# EPICS substitutions: odmApp/Db/odm-test.substitutions
file pilz-plc-bi-table9seg1.template
{
	pattern
	{dtype, areapos,  attribute,     description,                       port,    bit,   zname,         oname,                 zsv,        osv, plc           }

#################################################################### ODM PILZ PLC ##########################################################################

	{ ODM, CR1:1:0,  FAULT,         "C1 West Oxigraf Ch0 Real",       ODM_RD,      7,   OK,            FAULT,               NO_ALARM,   MAJOR, PLC:CP00:OD01 }
	{ ODM, CR1:1:0,  FAULT_LTH,     "C1 West Oxigraf Ch0 Latch",      ODM_RD,      6,   OK,            FAULT,               NO_ALARM,   MAJOR, PLC:CP00:OD01 }
	{ ODM, CR1:1:1,  FAULT,         "C1 West Oxigraf Ch1 Real",       ODM_RD,      5,   OK,            FAULT,               NO_ALARM,   MAJOR, PLC:CP00:OD01 }
	{ ODM, CR1:1:1,  FAULT_LTH,     "C1 West Oxigraf Ch1 Latch",      ODM_RD,      4,   OK,            FAULT,               NO_ALARM,   MAJOR, PLC:CP00:OD01 }
	{ ODM, CR1:1:2,  FAULT,         "C1 West Oxigraf Ch2 Real",       ODM_RD,      3,   OK,            FAULT,               NO_ALARM,   MAJOR, PLC:CP00:OD01 }
	{ ODM, CR1:1:2,  FAULT_LTH,     "C1 West Oxigraf Ch2 Latch",      ODM_RD,      2,   OK,            FAULT,               NO_ALARM,   MAJOR, PLC:CP00:OD01 }
	{ ODM, CR1:1:3,  FAULT,         "C1 West Oxigraf Ch3 Real",       ODM_RD,      1,   OK,            FAULT,               NO_ALARM,   MAJOR, PLC:CP00:OD01 }
	{ ODM, CR1:1:3,  FAULT_LTH,     "C1 West Oxigraf Ch3 Latch",      ODM_RD,      0,   OK,            FAULT,               NO_ALARM,   MAJOR, PLC:CP00:OD01 }
	{ ODM, CR1:2:0,  FAULT,         "C1 East Oxigraf Ch0 Real",       ODM_RD,      15,  OK,            FAULT,               NO_ALARM,   MAJOR, PLC:CP00:OD01 }
	{ ODM, CR1:2:0,  FAULT_LTH,     "C1 East Oxigraf Ch0 Latch",      ODM_RD,      14,  OK,            FAULT,               NO_ALARM,   MAJOR, PLC:CP00:OD01 }
	{ ODM, CR1:2:1,  FAULT,         "C1 East Oxigraf Ch1 Real",       ODM_RD,      13,  OK,            FAULT,               NO_ALARM,   MAJOR, PLC:CP00:OD01 }
	{ ODM, CR1:2:1,  FAULT_LTH,     "C1 East Oxigraf Ch1 Latch",      ODM_RD,      12,  OK,            FAULT,               NO_ALARM,   MAJOR, PLC:CP00:OD01 }
	{ ODM, CR1:2:2,  FAULT,         "C1 East Oxigraf Ch2 Real",       ODM_RD,      11,  OK,            FAULT,               NO_ALARM,   MAJOR, PLC:CP00:OD01 }
	{ ODM, CR1:2:2,  FAULT_LTH,     "C1 East Oxigraf Ch2 Latch",      ODM_RD,      10,  OK,            FAULT,               NO_ALARM,   MAJOR, PLC:CP00:OD01 }
	{ ODM, CR1:2:3,  FAULT,         "C1 East Oxigraf Ch3 Real",       ODM_RD,      9,   OK,            FAULT,               NO_ALARM,   MAJOR, PLC:CP00:OD01 }
	{ ODM, CR1:2:3,  FAULT_LTH,     "C1 East Oxigraf Ch3 Latch",      ODM_RD,      8,   OK,            FAULT,               NO_ALARM,   MAJOR, PLC:CP00:OD01 }
	{ ODM, CR1:1,    SYS_OK,        "C1 West Sys OK Real",            ODM_RD,      23,  OK,            FAULT,               NO_ALARM,   MAJOR, PLC:CP00:OD01 }
	{ ODM, CR1:1,    SYS_OK_LTH,    "C1 West Sys OK Latch",           ODM_RD,      22,  OK,            FAULT,               NO_ALARM,   MAJOR, PLC:CP00:OD01 }
	{ ODM, CR1:2,    SYS_OK,        "C1 East Sys OK Real",            ODM_RD,      21,  OK,            FAULT,               NO_ALARM,   MAJOR, PLC:CP00:OD01 }
	{ ODM, CR1:2,    SYS_OK_LTH,    "C1 East Sys OK Latch",           ODM_RD,      20,  OK,            FAULT,               NO_ALARM,   MAJOR, PLC:CP00:OD01 }
	{ ODM, CR0:1:0,  FAULT,         "CBR West Oxigraf Ch0 Real",      ODM_RD,      19,  OK,            FAULT,               NO_ALARM,   MAJOR, PLC:CP00:OD01 }
	{ ODM, CR0:1:0,  FAULT_LTH,     "CBR West Oxigraf Ch0 Latch",     ODM_RD,      18,  OK,            FAULT,               NO_ALARM,   MAJOR, PLC:CP00:OD01 }
	{ ODM, CR0:1:1,  FAULT,         "CBR West Oxigraf Ch1 Real",      ODM_RD,      17,  OK,            FAULT,               NO_ALARM,   MAJOR, PLC:CP00:OD01 }
	{ ODM, CR0:1:1,  FAULT_LTH,     "CBR West Oxigraf Ch1 Latch",     ODM_RD,      16,  OK,            FAULT,               NO_ALARM,   MAJOR, PLC:CP00:OD01 }
	{ ODM, CR0:1:2,  FAULT,         "CBR West Oxigraf Ch2 Real",      ODM_RD,      95,  OK,            FAULT,               NO_ALARM,   MAJOR, PLC:CP00:OD01 }
	{ ODM, CR0:1:2,  FAULT_LTH,     "CBR West Oxigraf Ch2 Latch",     ODM_RD,      94,  OK,            FAULT,               NO_ALARM,   MAJOR, PLC:CP00:OD01 }
	{ ODM, CR0:1:3,  FAULT,         "CBR West Oxigraf Ch3 Real",      ODM_RD,      93,  OK,            FAULT,               NO_ALARM,   MAJOR, PLC:CP00:OD01 }
	{ ODM, CR0:1:3,  FAULT_LTH,     "CBR West Oxigraf Ch3 Latch",     ODM_RD,      92,  OK,            FAULT,               NO_ALARM,   MAJOR, PLC:CP00:OD01 }
	{ ODM, CR0:2:0,  FAULT,         "CBR East Oxigraf Ch0 Real",      ODM_RD,      91,  OK,            FAULT,               NO_ALARM,   MAJOR, PLC:CP00:OD01 }
	{ ODM, CR0:2:0,  FAULT_LTH,     "CBR East Oxigraf Ch0 Latch",     ODM_RD,      90,  OK,            FAULT,               NO_ALARM,   MAJOR, PLC:CP00:OD01 }
	{ ODM, CR0:2:1,  FAULT,         "CBR East Oxigraf Ch1 Real",      ODM_RD,      89,  OK,            FAULT,               NO_ALARM,   MAJOR, PLC:CP00:OD01 }
	{ ODM, CR0:2:1,  FAULT_LTH,     "CBR East Oxigraf Ch1 Latch",     ODM_RD,      88,  OK,            FAULT,               NO_ALARM,   MAJOR, PLC:CP00:OD01 }
	{ ODM, CR0:2:2,  FAULT,         "CBR East Oxigraf Ch2 Real",      ODM_RD,      103, OK,            FAULT,               NO_ALARM,   MAJOR, PLC:CP00:OD01 }
	{ ODM, CR0:2:2,  FAULT_LTH,     "CBR East Oxigraf Ch2 Latch",     ODM_RD,      102, OK,            FAULT,               NO_ALARM,   MAJOR, PLC:CP00:OD01 }
	{ ODM, CR0:2:3,  FAULT,         "CBR East Oxigraf Ch3 Real",      ODM_RD,      101, OK,            FAULT,               NO_ALARM,   MAJOR, PLC:CP00:OD01 }
	{ ODM, CR0:2:3,  FAULT_LTH,     "CBR East Oxigraf Ch3 Latch",     ODM_RD,      100, OK,            FAULT,               NO_ALARM,   MAJOR, PLC:CP00:OD01 }
	{ ODM, CR0:1,    SYS_OK,        "CBR West Sys OK Real",           ODM_RD,      99,  OK,            FAULT,               NO_ALARM,   MAJOR, PLC:CP00:OD01 }
	{ ODM, CR0:1,    SYS_OK_LTH,    "CBR West Sys OK Latch",          ODM_RD,      98,  OK,            FAULT,               NO_ALARM,   MAJOR, PLC:CP00:OD01 }
	{ ODM, CR0:2,    SYS_OK,        "CBR East Sys OK Real",           ODM_RD,      97,  OK,            FAULT,               NO_ALARM,   MAJOR, PLC:CP00:OD01 }
	{ ODM, CR0:2,    SYS_OK_LTH,    "CBR East Sys OK Latch",          ODM_RD,      96,  OK,            FAULT,               NO_ALARM,   MAJOR, PLC:CP00:OD01 }
	{ ODM, CR2:1:0,  FAULT,         "C2 West Oxigraf Ch0 Real",       ODM_RD,      111, OK,            FAULT,               NO_ALARM,   MAJOR, PLC:CP00:OD01 }
	{ ODM, CR2:1:0,  FAULT_LTH,     "C2 West Oxigraf Ch0 Latch",      ODM_RD,      110, OK,            FAULT,               NO_ALARM,   MAJOR, PLC:CP00:OD01 }
	{ ODM, CR2:1:1,  FAULT,         "C2 West Oxigraf Ch1 Real",       ODM_RD,      109, OK,            FAULT,               NO_ALARM,   MAJOR, PLC:CP00:OD01 }
	{ ODM, CR2:1:1,  FAULT_LTH,     "C2 West Oxigraf Ch1 Latch",      ODM_RD,      108, OK,            FAULT,               NO_ALARM,   MAJOR, PLC:CP00:OD01 }
	{ ODM, CR2:1:2,  FAULT,         "C2 West Oxigraf Ch2 Real",       ODM_RD,      107, OK,            FAULT,               NO_ALARM,   MAJOR, PLC:CP00:OD01 }
	{ ODM, CR2:1:2,  FAULT_LTH,     "C2 West Oxigraf Ch2 Latch",      ODM_RD,      106, OK,            FAULT,               NO_ALARM,   MAJOR, PLC:CP00:OD01 }
	{ ODM, CR2:1:3,  FAULT,         "C2 West Oxigraf Ch3 Real",       ODM_RD,      105, OK,            FAULT,               NO_ALARM,   MAJOR, PLC:CP00:OD01 }
	{ ODM, CR2:1:3,  FAULT_LTH,     "C2 West Oxigraf Ch3 Latch",      ODM_RD,      104, OK,            FAULT,               NO_ALARM,   MAJOR, PLC:CP00:OD01 }
	{ ODM, CR2:2:0,  FAULT,         "C2 East Oxigraf Ch0 Real",       ODM_RD,      119, OK,            FAULT,               NO_ALARM,   MAJOR, PLC:CP00:OD01 }
	{ ODM, CR2:2:0,  FAULT_LTH,     "C2 East Oxigraf Ch0 Latch",      ODM_RD,      118, OK,            FAULT,               NO_ALARM,   MAJOR, PLC:CP00:OD01 }
	{ ODM, CR2:2:1,  FAULT,         "C2 East Oxigraf Ch1 Real",       ODM_RD,      117, OK,            FAULT,               NO_ALARM,   MAJOR, PLC:CP00:OD01 }
	{ ODM, CR2:2:1,  FAULT_LTH,     "C2 East Oxigraf Ch1 Latch",      ODM_RD,      116, OK,            FAULT,               NO_ALARM,   MAJOR, PLC:CP00:OD01 }
	{ ODM, CR2:2:2,  FAULT,         "C2 East Oxigraf Ch2 Real",       ODM_RD,      115, OK,            FAULT,               NO_ALARM,   MAJOR, PLC:CP00:OD01 }
	{ ODM, CR2:2:2,  FAULT_LTH,     "C2 East Oxigraf Ch2 Latch",      ODM_RD,      114, OK,            FAULT,               NO_ALARM,   MAJOR, PLC:CP00:OD01 }
	{ ODM, CR2:2:3,  FAULT,         "C2 East Oxigraf Ch3 Real",       ODM_RD,      113, OK,            FAULT,               NO_ALARM,   MAJOR, PLC:CP00:OD01 }
	{ ODM, CR2:2:3,  FAULT_LTH,     "C2 East Oxigraf Ch3 Latch",      ODM_RD,      112, OK,            FAULT,               NO_ALARM,   MAJOR, PLC:CP00:OD01 }
	{ ODM, CR2:1,    SYS_OK,        "C2 West Sys OK Real",            ODM_RD,      127, OK,            FAULT,               NO_ALARM,   MAJOR, PLC:CP00:OD01 }
	{ ODM, CR2:1,    SYS_OK_LTH,    "C2 West Sys OK Latch",           ODM_RD,      126, OK,            FAULT,               NO_ALARM,   MAJOR, PLC:CP00:OD01 }
	{ ODM, CR2:2,    SYS_OK,        "C2 East Sys OK Real",            ODM_RD,      125, OK,            FAULT,               NO_ALARM,   MAJOR, PLC:CP00:OD01 }
	{ ODM, CR2:2,    SYS_OK_LTH,    "C2 East Sys OK Latch",           ODM_RD,      124, OK,            FAULT,               NO_ALARM,   MAJOR, PLC:CP00:OD01 }
	{ ODM, CR1,      AC_OK     ,    "C1 AC OK Sum",                   ODM_RD,      123, "AC OK",       "AC Not OK",         NO_ALARM,   MAJOR, PLC:CP00:OD01 }
	{ ODM, CR1,      AL_MUTED,      "C1 Alarm Mute",                  ODM_RD,      122, NOT_MUTED,     MUTED,               NO_ALARM,   MINOR, PLC:CP00:OD01 }
	{ ODM, CR1,      STROBE,        "C1 Strobe Out",                  ODM_RD,      121, STROBE_OFF,    STROBE_ON,           NO_ALARM,NO_ALARM, PLC:CP00:OD01 }
	{ ODM, CR1,      HORN,          "C1 Horn Out",                    ODM_RD,      120, HORN_OFF,      HORN_ON,             NO_ALARM,NO_ALARM, PLC:CP00:OD01 }
	{ ODM, CR1,      FAN,           "C1 Fan Out",                     ODM_RD,      135, FAN_OFF,       FAN_ON,              NO_ALARM,NO_ALARM, PLC:CP00:OD01 }
	{ ODM, CR0,      AC_OK     ,    "CB AC OK Sum",                   ODM_RD,      134, "AC OK",       "AC Not OK",         NO_ALARM,   MAJOR, PLC:CP00:OD01 }
	{ ODM, CR1:1,    OXGF_DISABLED, "C1 West Oxigraf Disable",        ODM_RD,      133, ENABLED,       DISABLED,            NO_ALARM,   MINOR, PLC:CP00:OD01 }
	{ ODM, CR1:2,    OXGF_DISABLED, "C1 East Oxigraf Disable",        ODM_RD,      132, ENABLED,       DISABLED,            NO_ALARM,   MINOR, PLC:CP00:OD01 }
	{ ODM, CR2,      AC_OK     ,    "C2 AC OK Sum",                   ODM_RD,      131, "AC OK",       "AC Not OK",         NO_ALARM,   MAJOR, PLC:CP00:OD01 }
	{ ODM, CR0,      AL_MUTED,      "CBR Alarm Mute",                 ODM_RD,      130, NOT_MUTED,     MUTED,               NO_ALARM,   MINOR, PLC:CP00:OD01 }
	{ ODM, CR0,      STROBE,        "CBR Strobe Out",                 ODM_RD,      129, STROBE_OFF,    STROBE_ON,           NO_ALARM,NO_ALARM, PLC:CP00:OD01 }
	{ ODM, CR0,      HORN,          "CBR Horn Out",                   ODM_RD,      128, HORN_OFF,      HORN_ON,             NO_ALARM,NO_ALARM, PLC:CP00:OD01 }
	{ ODM, CR0,      FAN,           "CBR Fan Out",                    ODM_RD,      143, FAN_OFF,       FAN_ON,              NO_ALARM,NO_ALARM, PLC:CP00:OD01 }
	{ ODM, CP00:1,   TEST_MODE,     "TRI Test Mode Key Switch",       ODM_RD,      142, Normal,        Test,                NO_ALARM,   MAJOR, PLC:CP00:OD01 }
	{ ODM, CR0:1,    OXGF_DISABLE,  "CBR West Oxigraf Disable",       ODM_RD,      141, ENABLED,       DISABLED,            NO_ALARM,   MINOR, PLC:CP00:OD01 }
	{ ODM, CR0:2,    OXGF_DISABLE,  "CBR East Oxigraf Disable",       ODM_RD,      140, ENABLED,       DISABLED,            NO_ALARM,   MINOR, PLC:CP00:OD01 }
	{ ODM, CP00:1,   DC_OK,         "DC power supply PS1 Ok",         ODM_RD,      139, FAULT,         OK,                  MAJOR,   NO_ALARM, PLC:CP00:OD01 }
	{ ODM, CR2,      AL_MUTE,       "C2 Alarm Mute",                  ODM_RD,      138, NOT_MUTED,     MUTED,               NO_ALARM,   MINOR, PLC:CP00:OD01 }
	{ ODM, CR2,      STROBE,        "C2 Strobe Out",                  ODM_RD,      137, STROBE_OFF,    STROBE_ON,           NO_ALARM,NO_ALARM, PLC:CP00:OD01 }
	{ ODM, CR2,      HORN,          "C2 Horn Out",                    ODM_RD,      136, HORN_OFF,      HORN_ON,             NO_ALARM,NO_ALARM, PLC:CP00:OD01 }
	{ ODM, CR2,      FAN,           "C2 Fan Out",                     ODM_RD,      151, FAN_OFF,       FAN_ON,              NO_ALARM,NO_ALARM, PLC:CP00:OD01 }
	{ ODM, CP00:2,   DC_OK,         "DC power supply PS2 Ok",         ODM_RD,      150, FAULT,         OK,                  MAJOR,   NO_ALARM, PLC:CP00:OD01 }
	{ ODM, CR2:1,    OXGF_DISABLE,  "C2 West Oxigraf Disable",        ODM_RD,      149, ENABLED,       DISABLED,            NO_ALARM,   MINOR, PLC:CP00:OD01 }
	{ ODM, CR2:2,    OXGF_DISABLE,  "C2 East Oxigraf Disable",        ODM_RD,      148, ENABLED,       DISABLED,            NO_ALARM,   MINOR, PLC:CP00:OD01 }
#	level 1 alarm
	{ ODM, CP00,     YELLOW_ALARM,  "Yellow Alarm",                   ODM_RD,      147, NO_YELLOW_ALARM,YELLOW_ALARM,       NO_ALARM,   MINOR, PLC:CP00:OD01 }
#	level 2 alarm
	{ ODM, CP00,     RED_ALARM,     "Red Alarm",                      ODM_RD,      146, NO_RED_ALARM,  RED_ALARM,           NO_ALARM,   MAJOR, PLC:CP00:OD01 }
	{ ODM, CP00,     HEARTBEAT,     "PLC Heart Beat",                 ODM_RD,      145, LOW,           HIGH,                MAJOR,   NO_ALARM, PLC:CP00:OD01 }
	{ ODM, CP00,     ACR_ALARM,     "ACR Alarm",                      ODM_RD,      144, NO_ACR_ALARM,  ACR_ALARM,           NO_ALARM,   MAJOR, PLC:CP00:OD01 }

}

file pilz-plc-bo.template
{
	pattern
	{dtype,areapos,  attribute,            description,                      port,      bit,   zname,            oname,            zsv,     osv      }
	{ ODM, CR1:1,    SET_OXGF_DISABLE,     "C1 West Oxigraf Disable",        ODM_WRT,     7,   NOT_DISABLE,      DISABLE,          NO_ALARM,NO_ALARM }
	{ ODM, CR1:1,    SET_OXGF_ENABLE,      "C1 West Oxigraf Enable",         ODM_WRT,     6,   NOT_ENABLE,       ENABLE,           NO_ALARM,NO_ALARM }
	{ ODM, CR1:2,    SET_OXGF_DISABLE,     "C1 East Oxigraf Disable",        ODM_WRT,     5,   NOT_DISABLE,      DISABLE,          NO_ALARM,NO_ALARM }
	{ ODM, CR1:2,    SET_OXGF_ENABLE,      "C1 East Oxigraf Enable",         ODM_WRT,     4,   NOT_ENABLE,       ENABLE,           NO_ALARM,NO_ALARM }
	{ ODM, CR0:1,    SET_OXGF_DISABLE,     "CBR West Oxigraf Disable",       ODM_WRT,     3,   NOT_DISABLE,      DISABLE,          NO_ALARM,NO_ALARM }
	{ ODM, CR0:1,    SET_OXGF_ENABLE,      "CBR West Oxigraf Enable",        ODM_WRT,     2,   NOT_ENABLE,       ENABLE,           NO_ALARM,NO_ALARM }
	{ ODM, CR0:2,    SET_OXGF_DISABLE,     "CBR East Oxigraf Disable",       ODM_WRT,     1,   NOT_DISABLE,      DISABLE,          NO_ALARM,NO_ALARM }
	{ ODM, CR0:2,    SET_OXGF_ENABLE,      "CBR East Oxigraf Enable",        ODM_WRT,     0,   NOT_ENABLE,       ENABLE,           NO_ALARM,NO_ALARM }
	{ ODM, CR2:1,    SET_OXGF_DISABLE,     "C2 West Oxigraf Disable",        ODM_WRT,     15,  NOT_DISABLE,      DISABLE,          NO_ALARM,NO_ALARM }
	{ ODM, CR2:1,    SET_OXGF_ENABLE,      "C2 West Oxigraf Enable",         ODM_WRT,     14,  NOT_ENABLE,       ENABLE,           NO_ALARM,NO_ALARM }
	{ ODM, CR2:2,    SET_OXGF_DISABLE,     "C2 East OxigrafDisable",         ODM_WRT,     13,  NOT_DISABLE,      DISABLE,          NO_ALARM,NO_ALARM }
	{ ODM, CR2:2,    SET_OXGF_ENABLE,      "C2 East Oxigraf Enable",         ODM_WRT,     12,  NOT_ENABLE,       ENABLE,           NO_ALARM,NO_ALARM }
	{ ODM, CP00,     SET_AL_RESET,         "Alarm Reset",                    ODM_WRT,     11,  NOT_RESET,        RESET,            NO_ALARM,NO_ALARM }
	{ ODM, CR1,      SET_AL_MUTE,          "C1 Alarm Mute",                  ODM_WRT,     9,   NOT_MUTE,         MUTE,             NO_ALARM,NO_ALARM }
	{ ODM, CR1,      SET_FAN_FORCE,        "C1 Fan Force",                   ODM_WRT,     8,   NOT_FAN_FORCE,    FAN_FORCE,        NO_ALARM,NO_ALARM }
	{ ODM, CR0,      SET_AL_MUTE,          "CBR Alarm Mute",                 ODM_WRT,     21,  NOT_MUTE,         MUTE,             NO_ALARM,NO_ALARM }
	{ ODM, CR0,      SET_FAN_FORCE,        "CBR Fan Force",                  ODM_WRT,     20,  NOT_FAN_FORCE,    FAN_FORCE,        NO_ALARM,NO_ALARM }
	{ ODM, CR2,      SET_AL_MUTE,          "C2 Alarm Mute",                  ODM_WRT,     17,  NOT_MUTE,         MUTE,             NO_ALARM,NO_ALARM }
	{ ODM, CR2,      SET_FAN_FORCE,        "C2 Fan Force",                   ODM_WRT,     16,  NOT_FAN_FORCE,    FAN_FORCE,        NO_ALARM,NO_ALARM }
}

file "pilz-plc-request.template"
{
	pattern
	{dtype,areapos,   port_rd, port_wrt  }
	{PLC,CP00:OD01,   ODM_RD,  ODM_WRT   }
}

file "pilz-plc-checksum.template"
{
        pattern
        {dtype,areapos,        port   }
        {PLC,  CP00:OD01,      ODM_WD }
}

file "statistics.template"
{ pattern
{P,                    R,      PORT,          SCAN}
{PLC:CP00:OD01,  :ODM_RD,    ODM_RD,   "10 second"}
{PLC:CP00:OD01,  :ODM_WRT,   ODM_WRT,  "10 second"}
{PLC:CP00:OD01,  :ODM_WD,    ODM_WD,   "10 second"}
}

file asynRecord.db
{
pattern{ P               , R          , PORT, ADDR, IMAX, OMAX }
		{ PLC:CP00:OD01: , ASYNDRIVER , ODM , 0,0, 0    }
}

#file MO2i.template
#{
#pattern	{ PRIM, LOCA, UNIT, PORT,                SCAN      }
#		{ ODM,  CR1,  1,    OXI_$(LOCA)$(UNIT), "1 second" }
#		{ ODM,  CR1,  2,    OXI_$(LOCA)$(UNIT), "1 second" }
#		{ ODM,  CR0,  1,    OXI_$(LOCA)$(UNIT), "1 second" }
#		{ ODM,  CR0,  2,    OXI_$(LOCA)$(UNIT), "1 second" }
#		{ ODM,  CR2,  1,    OXI_$(LOCA)$(UNIT), "1 second" }
#		{ ODM,  CR2,  2,    OXI_$(LOCA)$(UNIT), "1 second" }
#}
#
#file asynRecord.db
#{
#pattern{ P               , R          , PORT, ADDR, IMAX, OMAX }
#		{ SIOC:CP00:OD01:, ASYNDRIVER , OXI_CR11,  0,0, 0    }
#}
